ABB RobotStudio station: Project3.rsstnx

Station Project3 (saved by RobotStudio 25.4.11475.0)
Controller IRB140_6_81, task T_ROB1: task frame (RAPID world) sits at (0, 0, 400) mm in the station
Controller IRB140_6_81
  mechanical unit ROB_1: IRB140_6_81_C_03, 6 joints, base frame (0, 0, 0) mm
Layout (positions relative to the parent item):
  - IRB140_6_81_C_03 [mechanism, from %ABB.RobotStudio.Models.IRB140%\IRB140_6_81_C_G_03.rslib] at (0, 0, 400) mm; joint values [0, 0, 0, 0, 0, 0] (rad or m)
  - Pedestal [part], size 468 x 422 x 400 mm
  - Mesa [part] at (0, 0, 0) mm, rotated rx 90 ry 0 rz 90 deg, size 400 x 675 x 615 mm
  - Banda tranportadora [part], size 280 x 3100 x 448 mm
  - pcb [part] at (-260, -440, -40) mm, rotated rx 0 ry 0 rz 90 deg, size 51 x 70 x 12 mm
  - pcb_2 [part] at (-260, -650, -40) mm, rotated rx 0 ry 0 rz 90 deg, size 51 x 70 x 12 mm
  - gripper [mechanism] at (515, 0, 1112) mm, rotated rx 0 ry 90 rz 0 deg
      TCP gripperTCP1 at (6.14, 21.22, 139.97) mm
      TCP gripperTCP2 at (6.06, -18.4, 139.75) mm
      links: gripper2
  - caja [part] at (527, 0, 443) mm, rotated rx 90 ry 0 rz -90 deg, size 255 x 35 x 192 mm
Attachment: gripper is attached to IRB140_6_81_C_03 / Link6
Targets, tools, work objects and paths stored in the station, written as RAPID:
! task T_ROB1
MODULE CalibData
  PERS tooldata gripperTCP1:=[TRUE,[[6.141,21.217,139.967],[1,0,0,0]],[1,[0,0,1],[1,0,0,0],0,0,0]];
  PERS tooldata gripperTCP2:=[TRUE,[[6.063,-18.395,139.747],[1,0,0,0]],[1,[0,0,1],[1,0,0,0],0,0,0]];
ENDMODULE

! task T_ROB1
MODULE Module1
  PERS tooldata toolGripper:=[TRUE,[[5.679722754,2.287280651,120.075445417],[1,0,0,0]],[1,[0,0,1],[1,0,0,0],0,0,0]];
  PERS wobjdata wobj_Mesa:=[FALSE,TRUE,"",[[0,0,0],[1,0,0,0]],[[0,0,0],[1,0,0,0]]];
  PERS wobjdata wobj_Banda:=[FALSE,TRUE,"",[[0,0,0],[1,0,0,0]],[[0,0,0],[1,0,0,0]]];
  CONST jointtarget Home_ABS:=[[0,0,0,0,0,0],[9E+09,9E+09,9E+09,9E+09,9E+09,9E+09]];
  CONST num T_SONDEO:=2;
  CONST num T_CONVEYOR:=4.275;
  CONST num T_ESPERA_GRIP:=2;
  VAR bool bTimeout:=FALSE;
  CONST num T_GRIPPER:=0.5;
  CONST num T_CAL_BANDA:=5;
  CONST robtarget pPCB1Grab:=[[96,-439,296.51],[0,1,0,0],[-1,0,1,0],[9E+09,9E+09,9E+09,9E+09,9E+09,9E+09]];
  CONST robtarget pPCB1_Approach:=[[96,-439,376.51],[0,1,0,0],[-1,0,1,0],[9E+09,9E+09,9E+09,9E+09,9E+09,9E+09]];
  CONST robtarget pPCB2_Approach:=[[95.999978066,-549.00001315,376.509928967],[-0.000000003,1,-0.000000044,-0.000000001],[-1,-1,1,0],[9E+09,9E+09,9E+09,9E+09,9E+09,9E+09]];
  CONST robtarget pPCB2Grab:=[[96,-549,296.51],[0,1,0,0],[-1,0,-2,0],[9E+09,9E+09,9E+09,9E+09,9E+09,9E+09]];
  CONST robtarget pCajaPlace:=[[582,63.5,78],[0,0,1,0],[0,0,0,0],[9E+09,9E+09,9E+09,9E+09,9E+09,9E+09]];
  CONST robtarget pCajaApproach:=[[582,63.5,408],[0,0,1,0],[0,0,0,0],[9E+09,9E+09,9E+09,9E+09,9E+09,9E+09]];
  CONST num T_RETROCESO:=5;
  CONST num T_PASO:=5;
  PROC main()
    Inicializar;
    EsperarOrden;
  ENDPROC
  PROC EsperarOrden()
    EsperarLiberacion;
    IrAHome;
    EsperarLiberacion;
    IrAHome;
    CalibrarBanda;
    EsperarLiberacion;
    CicloEtapa4;
    WaitTime T_SONDEO;
  ENDPROC
  PROC CicloEtapa4()
    EsperarConfirmacion;
    PosicionarCaja;
    VerificarParada;
    VerificarParada;
    DepositarEnCaja;
    VerificarParada;
    IrAHome;
    SenalarDone;
  ENDPROC
  PROC SenalarDone()
    SetDO DO_01,1;
    WaitTime 0.25;
    SetDO DO_01,0;
    WaitTime 0.25;
  ENDPROC
  PROC EsperarLiberacion()
    WaitTime T_SONDEO;
  ENDPROC
  PROC VerificarParada()
    Reset FWD_Conveyor;
    Reset BWD_Conveyor;
    IrAHome;
    IrAHome;
    AbrirGripper;
  ENDPROC
  PROC AbrirGripper()
    SetDO DO_04,0;
  ENDPROC
  PROC CerrarSobrePCB()
    SetDO DO_04,1;
  ENDPROC
  PROC CerrarSobreCaja()
    SetDO DO_04,0;
    SetDO DO_05,1;
  ENDPROC
  PROC IrAHome()
    AbrirGripper;
    MoveAbsJ Home_ABS,v300,fine,toolGripper;
  ENDPROC
  PROC Inicializar()
    ConfL \On;
    ConfJ \On;
    SingArea \Off;
    AbrirGripper;
    IrAHome;
    Reset FWD_Conveyor;
    Reset BWD_Conveyor;
    CalibrarBanda;
  ENDPROC
  PROC CalibrarBanda()
    Reset FWD_Conveyor;
    Reset BWD_Conveyor;
    EsperarConfirmacion;
    Reset FWD_Conveyor;
    Set BWD_Conveyor;
    WaitTime T_RETROCESO;
    Reset BWD_Conveyor;
    EsperarConfirmacion;
  ENDPROC
  PROC DepositarEnCaja()
    MoveJ pCajaApproach,v300,z10,toolGripper\WObj:=wobj_Banda;
    MoveL pCajaPlace,v50,fine,toolGripper\WObj:=wobj_Banda;
    AbrirGripper;
    MoveL pCajaApproach,v100,fine,toolGripper\WObj:=wobj_Banda;
  ENDPROC
  PROC PosicionarCaja()
    Reset BWD_Conveyor;
    Set FWD_Conveyor;
    WaitTime T_PASO;
    Reset FWD_Conveyor;
  ENDPROC
  PROC EsperarConfirmacion()
    EsperarLiberacion;
    Set FWD_Conveyor;
    EsperarLiberacion;
  ENDPROC
ENDMODULE

